// TIA Portal project "2024" (V15.1)

(* hardware
DEVICE "S7300/ET200M station_1"  S7-300 station
   slot 0: "Rail_0"  Rail  6ES7 390-1***0-0AA0
   slot 2: "PLC_1"  CPU 314C-2 PN/DP  6ES7 314-6EH04-0AB0  V3.3
      slot 2: "PROFINET interface_1"  PN-IO
         slot 1: "Port_1"  Port
         slot 2: "Port_2"  Port
      slot 5: "DI 24/DO 16_1"  DI24/DO16
      slot 6: "AI 5/AO 2_1"  AI5/AO2
      slot 7: "Count_1"  Counter
      slot 8: "Positioning_1"  Positioning
   slot 4: "DO 8x24VDC/2A_1"  DO8 x 24VDC / 2A  6ES7 322-1BF01-0AA0
*)

// ===== PLC "PLC_1"  CPU 314C-2 PN/DP =====

VAR_GLOBAL   // PLC tag table "Default tag table"
   "F5" AT %I0.0 : Bool;
   "S3" AT %I0.1 : Bool;
   "S4" AT %I0.2 : Bool;
   "S5" AT %I0.3 : Bool;
   "S6" AT %I0.4 : Bool;
   "S7" AT %I0.5 : Bool;
   "S8" AT %I0.6 : Bool;
   "S9" AT %I0.7 : Bool;
   "S10" AT %I1.0 : Bool;
   "S11" AT %I1.1 : Bool;
   "S12" AT %I1.2 : Bool;
   "BP1" AT %I1.3 : Bool;
   "B1" AT %I1.4 : Bool;
   "B2" AT %I1.5 : Bool;
   "B3" AT %I1.6 : Bool;
   "B11" AT %I1.7 : Bool;
   "B12" AT %I2.0 : Bool;
   "B21" AT %I2.1 : Bool;
   "B22" AT %I2.2 : Bool;
   "B31" AT %I2.3 : Bool;
   "B32" AT %I2.4 : Bool;
   "Reserve1" AT %I2.5 : Bool;
   "Reserve2" AT %I2.6 : Bool;
   "F7" AT %I2.7 : Bool;
   "M11" AT %Q0.0 : Bool;
   "M12" AT %Q0.1 : Bool;
   "M21" AT %Q0.2 : Bool;
   "M22" AT %Q0.3 : Bool;
   "M31" AT %Q0.4 : Bool;
   "M32" AT %Q0.5 : Bool;
   "Reserve3" AT %Q0.6 : Bool;
   "Reserve4" AT %Q0.7 : Bool;
   "P32" AT %Q1.0 : Bool;
   "P33" AT %Q1.1 : Bool;
   "Reserve5" AT %Q1.2 : Bool;
   "P2" AT %Q1.3 : Bool;
   "P3" AT %Q1.4 : Bool;
   "P4" AT %Q1.5 : Bool;
   "P5" AT %Q1.6 : Bool;
   "P6" AT %Q1.7 : Bool;
   "P7" AT %Q2.0 : Bool;
   "P8" AT %Q2.1 : Bool;
   "P10" AT %Q2.2 : Bool;
   "P11" AT %Q2.3 : Bool;
   "P12" AT %Q2.4 : Bool;
   "P13" AT %Q2.5 : Bool;
   "P14" AT %Q2.6 : Bool;
   "P15" AT %Q2.7 : Bool;
END_VAR

DATA_BLOCK "G_Master_DB"   // DB1
{ S7_Optimized_Access := 'FALSE' }
VERSION : 0.1
// stored: InstanceOfName G_Master
"G_Master"
BEGIN
END_DATA_BLOCK

DATA_BLOCK "G_Pulse_DB"   // DB4
{ S7_Optimized_Access := 'FALSE' }
VERSION : 0.1
// stored: InstanceOfName G_Pulse
"G_Pulse"
BEGIN
END_DATA_BLOCK

DATA_BLOCK "G_Manual_DB"   // DB5
{ S7_Optimized_Access := 'FALSE' }
VERSION : 0.1
// stored: InstanceOfName G_Manual
"G_Manual"
BEGIN
END_DATA_BLOCK

DATA_BLOCK "G_Indicator_DB"   // DB6
{ S7_Optimized_Access := 'FALSE' }
VERSION : 0.1
// stored: InstanceOfName G_Indicator
"G_Indicator"
BEGIN
END_DATA_BLOCK

DATA_BLOCK "G_Auto_DB"   // DB13
{ S7_Optimized_Access := 'FALSE' }
VERSION : 0.1
// stored: InstanceOfName G_Auto
"G_Auto"
BEGIN
END_DATA_BLOCK

DATA_BLOCK "G_Output_DB"   // DB14
{ S7_Optimized_Access := 'FALSE' }
VERSION : 0.1
// stored: InstanceOfName G_Output
"G_Output"
BEGIN
END_DATA_BLOCK

FUNCTION_BLOCK "G_Master"   // FB1, FBD
{ S7_Optimized_Access := 'FALSE' }
VERSION : 0.1
   VAR_INPUT
      BP1 : Bool;
      F5 : Bool;
      F7 : Bool;
      S3 : Bool;
      S4 : Bool;
      "G_Auto.X500" : Bool;
      "G_Manual.X300" : Bool;
      Xung : Bool;
   END_VAR
   VAR_OUTPUT
      G_Manual : Bool;
      G_Auto : Bool;
      P3 : Bool;
      P32 : Bool;
   END_VAR
   VAR
      X1 : Bool;
      X2 : Bool;
      X3 : Bool;
      X4 : Bool;
      X5 : Bool;
      MA : Bool;
      MM : Bool;
   END_VAR
BEGIN

REGION Network 1
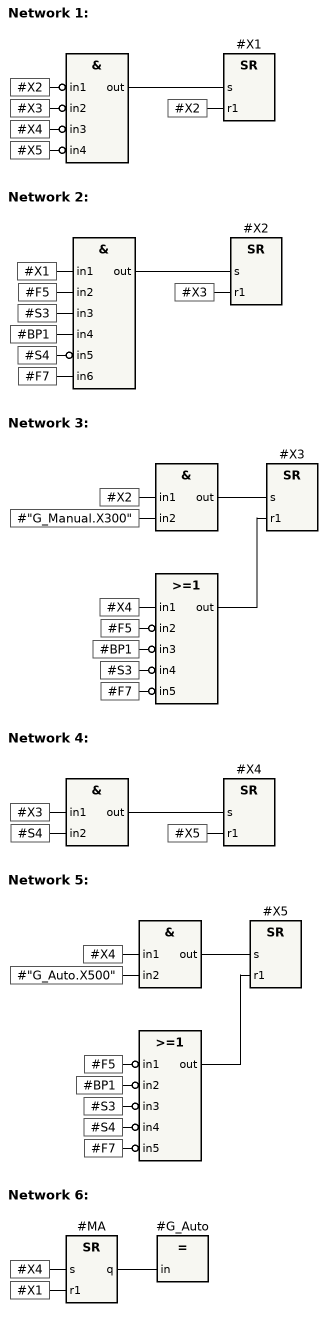
   IF NOT #X2 AND NOT #X3 AND NOT #X4 AND NOT #X5 THEN
       #X1 := TRUE;   // SR flip-flop
   END_IF;
   IF #X2 THEN #X1 := FALSE; END_IF;
END_REGION

REGION Network 2
   IF #X1 AND #F5 AND #S3 AND #BP1 AND NOT #S4 AND #F7 THEN
       #X2 := TRUE;   // SR flip-flop
   END_IF;
   IF #X3 THEN #X2 := FALSE; END_IF;
END_REGION

REGION Network 3
   IF #X2 AND #"G_Manual.X300" THEN
       #X3 := TRUE;   // SR flip-flop
   END_IF;
   IF #X4 OR NOT #F5 OR NOT #BP1 OR NOT #S3 OR NOT #F7 THEN #X3 := FALSE; END_IF;
END_REGION

REGION Network 4
   IF #X3 AND #S4 THEN
       #X4 := TRUE;   // SR flip-flop
   END_IF;
   IF #X5 THEN #X4 := FALSE; END_IF;
END_REGION

REGION Network 5
   IF #X4 AND #"G_Auto.X500" THEN
       #X5 := TRUE;   // SR flip-flop
   END_IF;
   IF NOT #F5 OR NOT #BP1 OR NOT #S3 OR NOT #S4 OR NOT #F7 THEN #X5 := FALSE; END_IF;
END_REGION

REGION Network 6
   IF #X4 THEN
       #MA := TRUE;   // SR flip-flop
   END_IF;
   IF #X1 THEN #MA := FALSE; END_IF;
   #G_Auto := #MA;
END_REGION

REGION Network 7
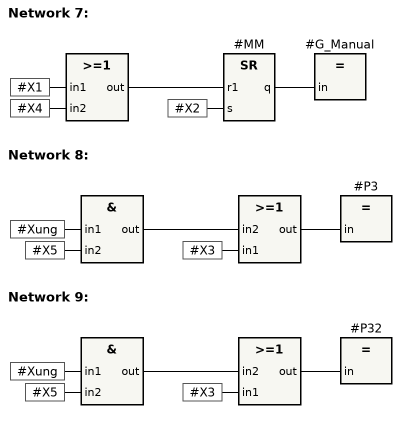
   IF #X2 THEN
       #MM := TRUE;   // SR flip-flop
   END_IF;
   IF #X1 OR #X4 THEN #MM := FALSE; END_IF;
   #G_Manual := #MM;
END_REGION

REGION Network 8
   #P3 := (#Xung AND #X5) OR #X3;
END_REGION

REGION Network 9
   #P32 := (#Xung AND #X5) OR #X3;
END_REGION
END_FUNCTION_BLOCK

FUNCTION_BLOCK "G_Pulse"   // FB2, FBD
{ S7_Optimized_Access := 'FALSE' }
VERSION : 0.1
   VAR_OUTPUT
      Pulse : Bool;
   END_VAR
   VAR
      X100 : Bool;
      X101 : Bool;
   END_VAR
BEGIN

REGION Network 1
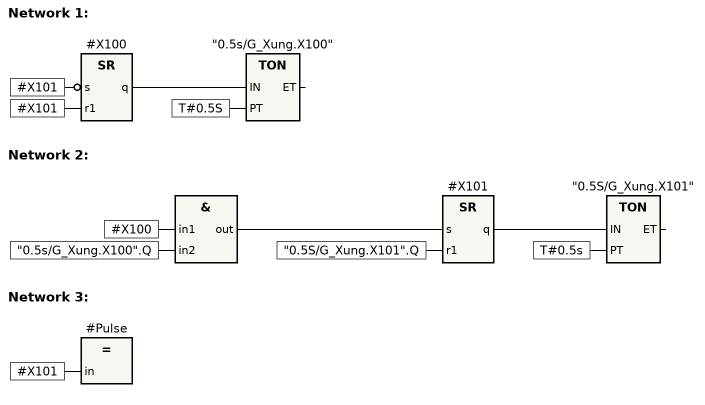
   IF NOT #X101 THEN
       #X100 := TRUE;   // SR flip-flop
   END_IF;
   IF #X101 THEN #X100 := FALSE; END_IF;
   "0.5s/G_Xung.X100".TON(IN := #X100, PT := T#0.5S);
END_REGION

REGION Network 2
   IF #X100 AND "0.5s/G_Xung.X100".Q THEN
       #X101 := TRUE;   // SR flip-flop
   END_IF;
   IF "0.5S/G_Xung.X101".Q THEN #X101 := FALSE; END_IF;
   "0.5S/G_Xung.X101".TON(IN := #X101, PT := T#0.5s);
END_REGION

REGION Network 3
   #Pulse := #X101;
END_REGION
END_FUNCTION_BLOCK

FUNCTION_BLOCK "G_Manual"   // FB3, FBD
{ S7_Optimized_Access := 'FALSE' }
VERSION : 0.1
   VAR_INPUT
      G_Manual : Bool;
      S4 : Bool;
      S6 : Bool;
      S7 : Bool;
      S8 : Bool;
      S9 : Bool;
      S10 : Bool;
      S11 : Bool;
   END_VAR
   VAR_OUTPUT
      M11 : Bool;
      M12 : Bool;
      M21 : Bool;
      M22 : Bool;
      M31 : Bool;
      M32 : Bool;
   END_VAR
   VAR
      X300 : Bool;
      X301 : Bool;
   END_VAR
BEGIN

REGION Network 1
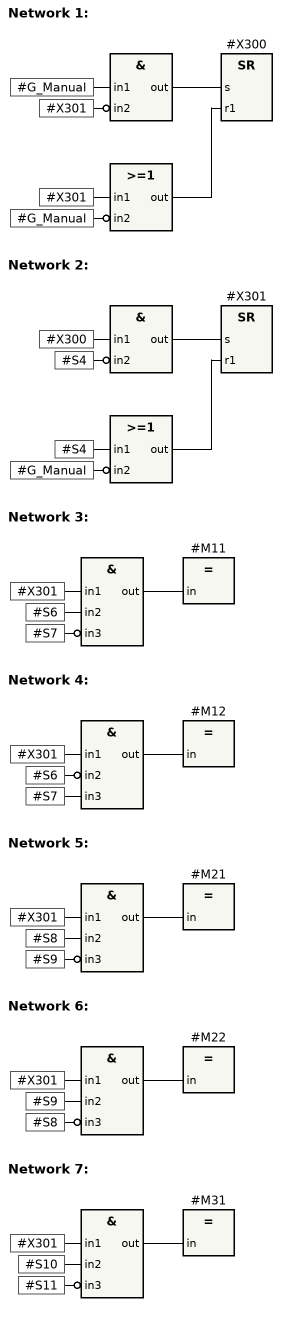
   IF #G_Manual AND NOT #X301 THEN
       #X300 := TRUE;   // SR flip-flop
   END_IF;
   IF #X301 OR NOT #G_Manual THEN #X300 := FALSE; END_IF;
END_REGION

REGION Network 2
   IF #X300 AND NOT #S4 THEN
       #X301 := TRUE;   // SR flip-flop
   END_IF;
   IF #S4 OR NOT #G_Manual THEN #X301 := FALSE; END_IF;
END_REGION

REGION Network 3
   #M11 := #X301 AND #S6 AND NOT #S7;
END_REGION

REGION Network 4
   #M12 := #X301 AND NOT #S6 AND #S7;
END_REGION

REGION Network 5
   #M21 := #X301 AND #S8 AND NOT #S9;
END_REGION

REGION Network 6
   #M22 := #X301 AND #S9 AND NOT #S8;
END_REGION

REGION Network 7
   #M31 := #X301 AND #S10 AND NOT #S11;
END_REGION

REGION Network 8
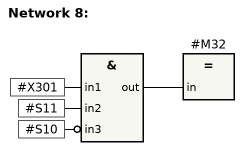
   #M32 := #X301 AND #S11 AND NOT #S10;
END_REGION
END_FUNCTION_BLOCK

FUNCTION_BLOCK "G_Indicator"   // FB4, FBD
{ S7_Optimized_Access := 'FALSE' }
VERSION : 0.1
   VAR_INPUT
      S3 : Bool;
      S12 : Bool;
      F7 : Bool;
      BP1 : Bool;
      B1 : Bool;
      B2 : Bool;
      B3 : Bool;
      B11 : Bool;
      B12 : Bool;
      B21 : Bool;
      B22 : Bool;
      B31 : Bool;
      B32 : Bool;
   END_VAR
   VAR_OUTPUT
      P2 : Bool;
      P3 : Bool;
      P4 : Bool;
      P5 : Bool;
      P6 : Bool;
      P7 : Bool;
      P8 : Bool;
      P10 : Bool;
      P11 : Bool;
      P12 : Bool;
      P13 : Bool;
      P14 : Bool;
      P15 : Bool;
      P32 : Bool;
      P33 : Bool;
   END_VAR
   VAR
      X200 : Bool;
      X201 : Bool;
   END_VAR
BEGIN

REGION Network 1
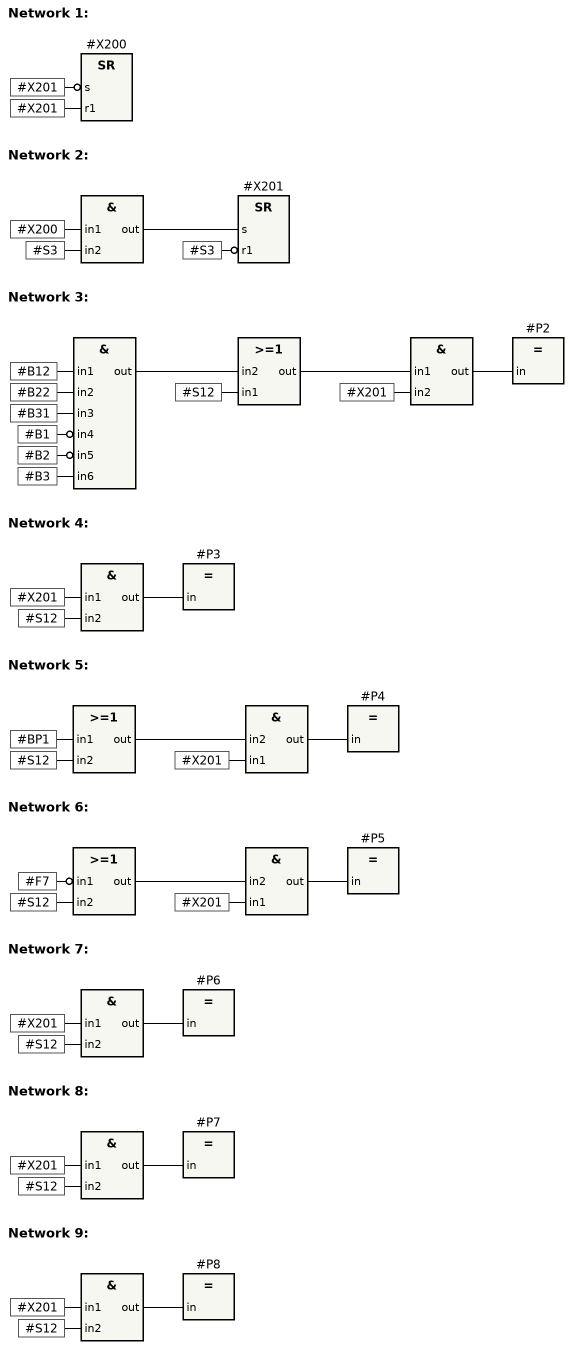
   IF NOT #X201 THEN
       #X200 := TRUE;   // SR flip-flop
   END_IF;
   IF #X201 THEN #X200 := FALSE; END_IF;
END_REGION

REGION Network 2
   IF #X200 AND #S3 THEN
       #X201 := TRUE;   // SR flip-flop
   END_IF;
   IF NOT #S3 THEN #X201 := FALSE; END_IF;
END_REGION

REGION Network 3
   #P2 := ((#B12 AND #B22 AND #B31 AND NOT #B1 AND NOT #B2 AND #B3) OR #S12) AND #X201;
END_REGION

REGION Network 4
   #P3 := #X201 AND #S12;
END_REGION

REGION Network 5
   #P4 := (#BP1 OR #S12) AND #X201;
END_REGION

REGION Network 6
   #P5 := (NOT #F7 OR #S12) AND #X201;
END_REGION

REGION Network 7
   #P6 := #X201 AND #S12;
END_REGION

REGION Network 8
   #P7 := #X201 AND #S12;
END_REGION

REGION Network 9
   #P8 := #X201 AND #S12;
END_REGION

REGION Network 10
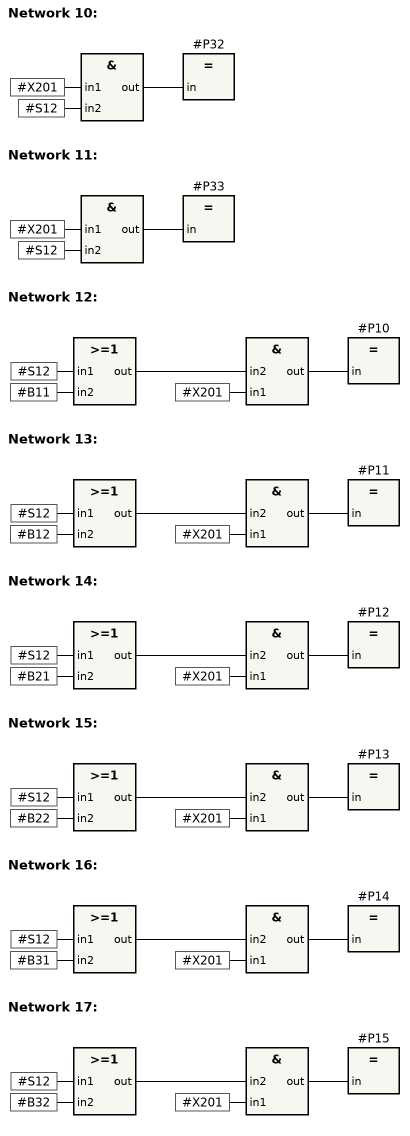
   #P32 := #X201 AND #S12;
END_REGION

REGION Network 11
   #P33 := #X201 AND #S12;
END_REGION

REGION Network 12
   #P10 := (#S12 OR #B11) AND #X201;
END_REGION

REGION Network 13
   #P11 := (#S12 OR #B12) AND #X201;
END_REGION

REGION Network 14
   #P12 := (#S12 OR #B21) AND #X201;
END_REGION

REGION Network 15
   #P13 := (#S12 OR #B22) AND #X201;
END_REGION

REGION Network 16
   #P14 := (#S12 OR #B31) AND #X201;
END_REGION

REGION Network 17
   #P15 := (#S12 OR #B32) AND #X201;
END_REGION
END_FUNCTION_BLOCK

FUNCTION_BLOCK "G_Auto"   // FB5, FBD
{ S7_Optimized_Access := 'FALSE' }
VERSION : 0.1
   VAR_INPUT
      "G_Master.X1" : Bool;
      G_Auto : Bool;
      S5 : Bool;
      B1 : Bool;
      B2 : Bool;
      B3 : Bool;
      B11 : Bool;
      B12 : Bool;
      B21 : Bool;
      B22 : Bool;
      B31 : Bool;
      B32 : Bool;
   END_VAR
   VAR_OUTPUT
      P6 : Bool;
      P7 : Bool;
      P8 : Bool;
      P33 : Bool;
      M11 : Bool;
      M12 : Bool;
      M21 : Bool;
      M22 : Bool;
      M31 : Bool;
      M32 : Bool;
   END_VAR
   VAR
      X500 : Bool;
      X501 : Bool;
      X502 : Bool;
      X503 : Bool;
      X503a : Bool;
      X504 : Bool;
      X504a : Bool;
      X505 : Bool;
      X506 : Bool;
      X507 : Bool;
      X508 : Bool;
      M6 : Bool;
      M7 : Bool;
   END_VAR
BEGIN

REGION Network 1
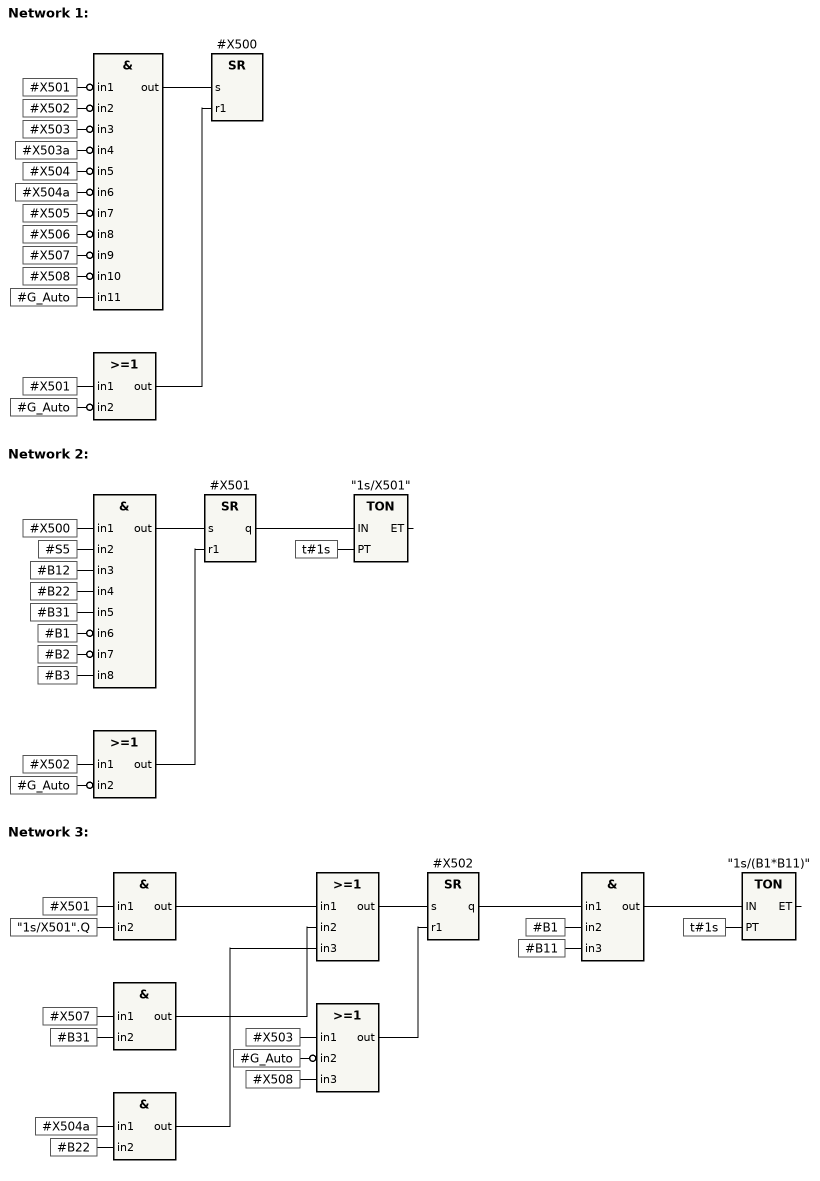
   IF NOT #X501 AND NOT #X502 AND NOT #X503 AND NOT #X503a AND NOT #X504 AND NOT #X504a AND NOT #X505 AND NOT #X506 AND NOT #X507 AND NOT #X508 AND #G_Auto THEN
       #X500 := TRUE;   // SR flip-flop
   END_IF;
   IF #X501 OR NOT #G_Auto THEN #X500 := FALSE; END_IF;
END_REGION

REGION Network 2
   IF #X500 AND #S5 AND #B12 AND #B22 AND #B31 AND NOT #B1 AND NOT #B2 AND #B3 THEN
       #X501 := TRUE;   // SR flip-flop
   END_IF;
   IF #X502 OR NOT #G_Auto THEN #X501 := FALSE; END_IF;
   "1s/X501".TON(IN := #X501, PT := t#1s);
END_REGION

REGION Network 3
   IF (#X501 AND "1s/X501".Q) OR (#X507 AND #B31) OR (#X504a AND #B22) THEN
       #X502 := TRUE;   // SR flip-flop
   END_IF;
   IF #X503 OR NOT #G_Auto OR #X508 THEN #X502 := FALSE; END_IF;
   "1s/(B1*B11)".TON(IN := #X502 AND #B1 AND #B11, PT := t#1s);
END_REGION

REGION Network 4
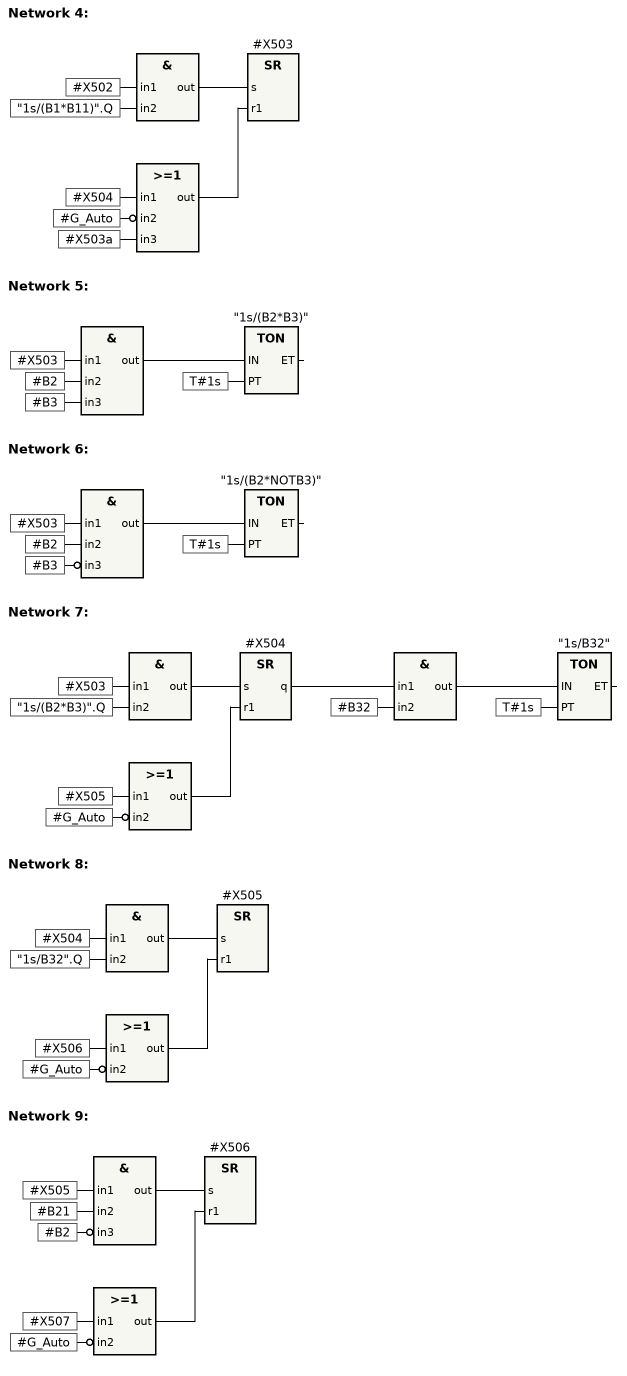
   IF #X502 AND "1s/(B1*B11)".Q THEN
       #X503 := TRUE;   // SR flip-flop
   END_IF;
   IF #X504 OR NOT #G_Auto OR #X503a THEN #X503 := FALSE; END_IF;
END_REGION

REGION Network 5
   "1s/(B2*B3)".TON(IN := #X503 AND #B2 AND #B3, PT := T#1s);
END_REGION

REGION Network 6
   "1s/(B2*NOTB3)".TON(IN := #X503 AND #B2 AND NOT #B3, PT := T#1s);
END_REGION

REGION Network 7
   IF #X503 AND "1s/(B2*B3)".Q THEN
       #X504 := TRUE;   // SR flip-flop
   END_IF;
   IF #X505 OR NOT #G_Auto THEN #X504 := FALSE; END_IF;
   "1s/B32".TON(IN := #X504 AND #B32, PT := T#1s);
END_REGION

REGION Network 8
   IF #X504 AND "1s/B32".Q THEN
       #X505 := TRUE;   // SR flip-flop
   END_IF;
   IF #X506 OR NOT #G_Auto THEN #X505 := FALSE; END_IF;
END_REGION

REGION Network 9
   IF #X505 AND #B21 AND NOT #B2 THEN
       #X506 := TRUE;   // SR flip-flop
   END_IF;
   IF #X507 OR NOT #G_Auto THEN #X506 := FALSE; END_IF;
END_REGION

REGION Network 10
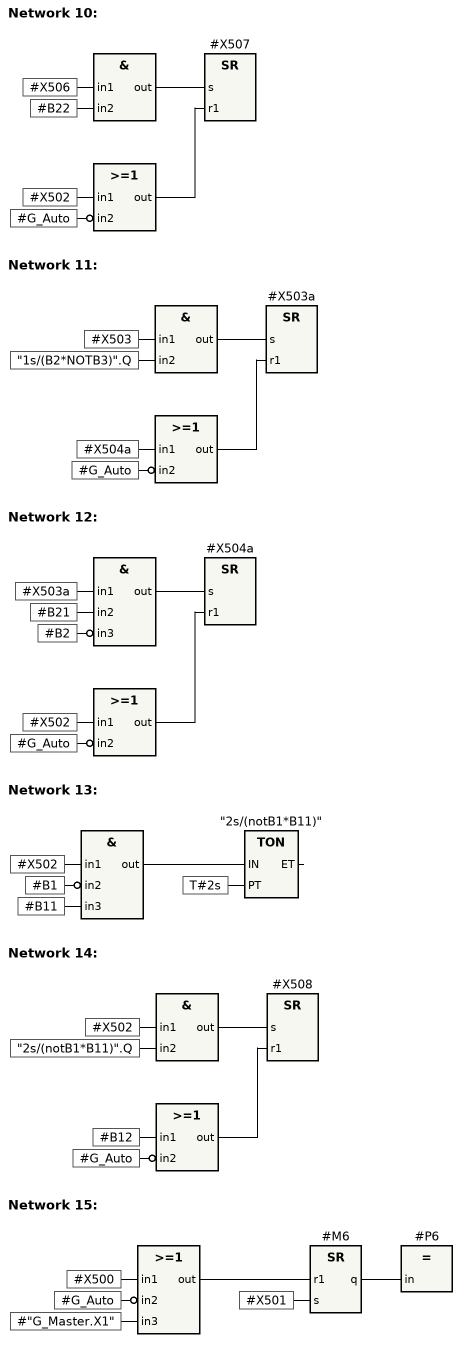
   IF #X506 AND #B22 THEN
       #X507 := TRUE;   // SR flip-flop
   END_IF;
   IF #X502 OR NOT #G_Auto THEN #X507 := FALSE; END_IF;
END_REGION

REGION Network 11
   IF #X503 AND "1s/(B2*NOTB3)".Q THEN
       #X503a := TRUE;   // SR flip-flop
   END_IF;
   IF #X504a OR NOT #G_Auto THEN #X503a := FALSE; END_IF;
END_REGION

REGION Network 12
   IF #X503a AND #B21 AND NOT #B2 THEN
       #X504a := TRUE;   // SR flip-flop
   END_IF;
   IF #X502 OR NOT #G_Auto THEN #X504a := FALSE; END_IF;
END_REGION

REGION Network 13
   "2s/(notB1*B11)".TON(IN := #X502 AND NOT #B1 AND #B11, PT := T#2s);
END_REGION

REGION Network 14
   IF #X502 AND "2s/(notB1*B11)".Q THEN
       #X508 := TRUE;   // SR flip-flop
   END_IF;
   IF #B12 OR NOT #G_Auto THEN #X508 := FALSE; END_IF;
END_REGION

REGION Network 15
   IF #X501 THEN
       #M6 := TRUE;   // SR flip-flop
   END_IF;
   IF #X500 OR NOT #G_Auto OR #"G_Master.X1" THEN #M6 := FALSE; END_IF;
   #P6 := #M6;
END_REGION

REGION Network 16
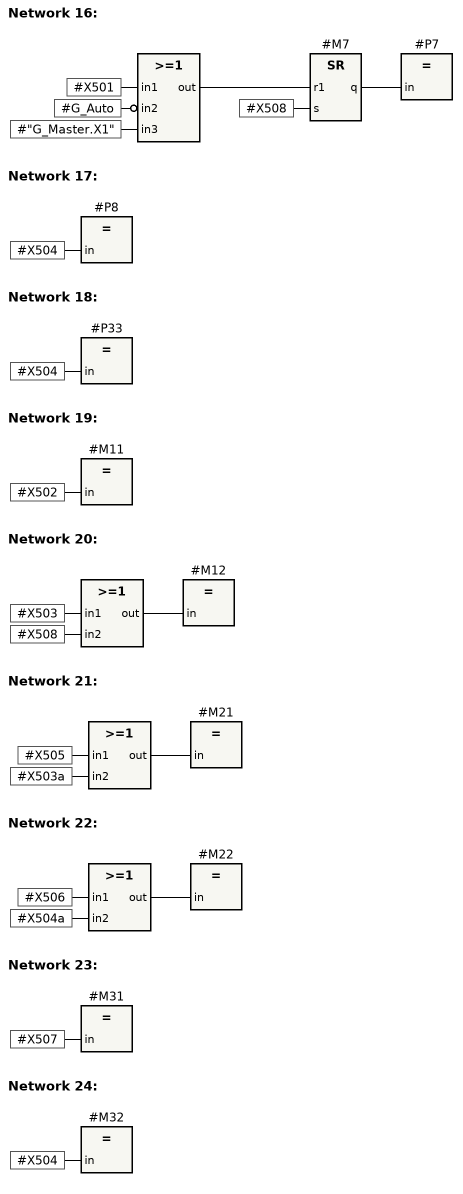
   IF #X508 THEN
       #M7 := TRUE;   // SR flip-flop
   END_IF;
   IF #X501 OR NOT #G_Auto OR #"G_Master.X1" THEN #M7 := FALSE; END_IF;
   #P7 := #M7;
END_REGION

REGION Network 17
   #P8 := #X504;
END_REGION

REGION Network 18
   #P33 := #X504;
END_REGION

REGION Network 19
   #M11 := #X502;
END_REGION

REGION Network 20
   #M12 := #X503 OR #X508;
END_REGION

REGION Network 21
   #M21 := #X505 OR #X503a;
END_REGION

REGION Network 22
   #M22 := #X506 OR #X504a;
END_REGION

REGION Network 23
   #M31 := #X507;
END_REGION

REGION Network 24
   #M32 := #X504;
END_REGION
END_FUNCTION_BLOCK

FUNCTION_BLOCK "G_Output"   // FB6, FBD
{ S7_Optimized_Access := 'FALSE' }
VERSION : 0.1
   VAR_INPUT
      M11_M : Bool;
      M12_M : Bool;
      M21_M : Bool;
      M22_M : Bool;
      M31_M : Bool;
      M32_M : Bool;
      M11_A : Bool;
      M12_A : Bool;
      M21_A : Bool;
      M22_A : Bool;
      M31_A : Bool;
      M32_A : Bool;
      P3_M : Bool;
      P32_M : Bool;
      P6_A : Bool;
      P7_A : Bool;
      P8_A : Bool;
      P33_A : Bool;
      P3_I : Bool;
      P6_I : Bool;
      P7_I : Bool;
      P8_I : Bool;
      P33_I : Bool;
      P32_I : Bool;
   END_VAR
   VAR_OUTPUT
      M11 : Bool;
      M12 : Bool;
      M21 : Bool;
      M22 : Bool;
      M31 : Bool;
      M32 : Bool;
      P3 : Bool;
      P6 : Bool;
      P7 : Bool;
      P8 : Bool;
      P33 : Bool;
      P32 : Bool;
   END_VAR
BEGIN

REGION Network 1
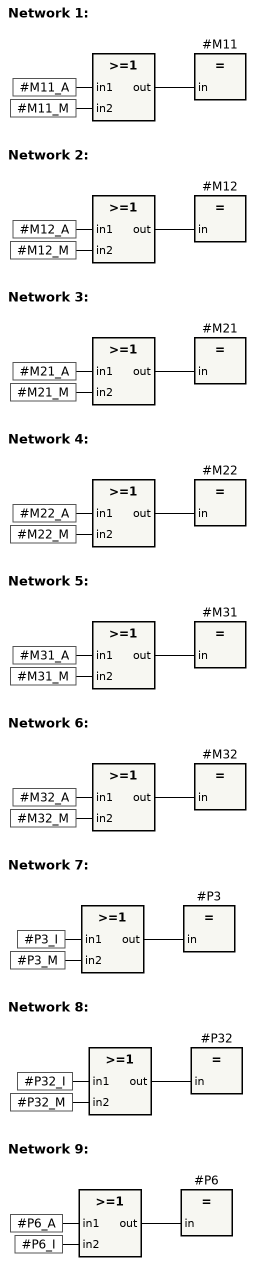
   #M11 := #M11_A OR #M11_M;
END_REGION

REGION Network 2
   #M12 := #M12_A OR #M12_M;
END_REGION

REGION Network 3
   #M21 := #M21_A OR #M21_M;
END_REGION

REGION Network 4
   #M22 := #M22_A OR #M22_M;
END_REGION

REGION Network 5
   #M31 := #M31_A OR #M31_M;
END_REGION

REGION Network 6
   #M32 := #M32_A OR #M32_M;
END_REGION

REGION Network 7
   #P3 := #P3_I OR #P3_M;
END_REGION

REGION Network 8
   #P32 := #P32_I OR #P32_M;
END_REGION

REGION Network 9
   #P6 := #P6_A OR #P6_I;
END_REGION

REGION Network 10
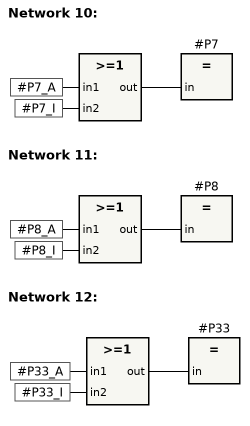
   #P7 := #P7_A OR #P7_I;
END_REGION

REGION Network 11
   #P8 := #P8_A OR #P8_I;
END_REGION

REGION Network 12
   #P33 := #P33_A OR #P33_I;
END_REGION
END_FUNCTION_BLOCK

ORGANIZATION_BLOCK "Main"   // OB1, FBD
TITLE = "Main Program Sweep (Cycle)"
{ S7_Optimized_Access := 'FALSE' }
VERSION : 0.1
   VAR_TEMP
      OB1_EV_CLASS : Byte;   // Bits 0-3 = 1 (Coming event), Bits 4-7 = 1 (Event class 1)
      OB1_SCAN_1 : Byte;   // 1 (Cold restart scan 1 of OB 1), 3 (Scan 2-n of OB 1)
      OB1_PRIORITY : Byte;   // Priority of OB Execution
      OB1_OB_NUMBR : Byte;   // 1 (Organization block 1, OB1)
      OB1_RESERVED_1 : Byte;   // Reserved for system
      OB1_RESERVED_2 : Byte;   // Reserved for system
      OB1_PREV_CYCLE : Int;   // Cycle time of previous OB1 scan (milliseconds)
      OB1_MIN_CYCLE : Int;   // Minimum cycle time of OB1 (milliseconds)
      OB1_MAX_CYCLE : Int;   // Maximum cycle time of OB1 (milliseconds)
      OB1_DATE_TIME : Date_And_Time;   // Date and time OB1 started
   END_VAR
BEGIN

REGION Network 1
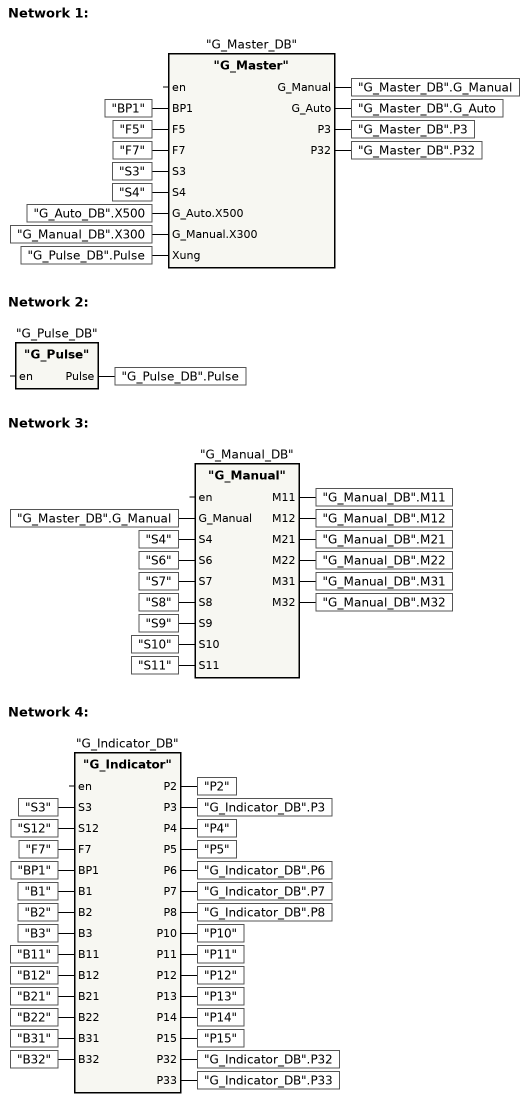
   "G_Master_DB"(BP1 := "BP1",   // "G_Master"
                 F5 := "F5",
                 F7 := "F7",
                 S3 := "S3",
                 S4 := "S4",
                 "G_Auto.X500" := "G_Auto_DB".X500,
                 "G_Manual.X300" := "G_Manual_DB".X300,
                 Xung := "G_Pulse_DB".Pulse,
                 G_Manual => "G_Master_DB".G_Manual,
                 G_Auto => "G_Master_DB".G_Auto,
                 P3 => "G_Master_DB".P3,
                 P32 => "G_Master_DB".P32);
END_REGION

REGION Network 2
   "G_Pulse_DB"(Pulse => "G_Pulse_DB".Pulse);   // "G_Pulse"
END_REGION

REGION Network 3
   "G_Manual_DB"(G_Manual := "G_Master_DB".G_Manual,   // "G_Manual"
                 S4 := "S4",
                 S6 := "S6",
                 S7 := "S7",
                 S8 := "S8",
                 S9 := "S9",
                 S10 := "S10",
                 S11 := "S11",
                 M11 => "G_Manual_DB".M11,
                 M12 => "G_Manual_DB".M12,
                 M21 => "G_Manual_DB".M21,
                 M22 => "G_Manual_DB".M22,
                 M31 => "G_Manual_DB".M31,
                 M32 => "G_Manual_DB".M32);
END_REGION

REGION Network 4
   "G_Indicator_DB"(S3 := "S3",   // "G_Indicator"
                    S12 := "S12",
                    F7 := "F7",
                    BP1 := "BP1",
                    B1 := "B1",
                    B2 := "B2",
                    B3 := "B3",
                    B11 := "B11",
                    B12 := "B12",
                    B21 := "B21",
                    B22 := "B22",
                    B31 := "B31",
                    B32 := "B32",
                    P2 => "P2",
                    P3 => "G_Indicator_DB".P3,
                    P4 => "P4",
                    P5 => "P5",
                    P6 => "G_Indicator_DB".P6,
                    P7 => "G_Indicator_DB".P7,
                    P8 => "G_Indicator_DB".P8,
                    P10 => "P10",
                    P11 => "P11",
                    P12 => "P12",
                    P13 => "P13",
                    P14 => "P14",
                    P15 => "P15",
                    P32 => "G_Indicator_DB".P32,
                    P33 => "G_Indicator_DB".P33);
END_REGION

REGION Network 5
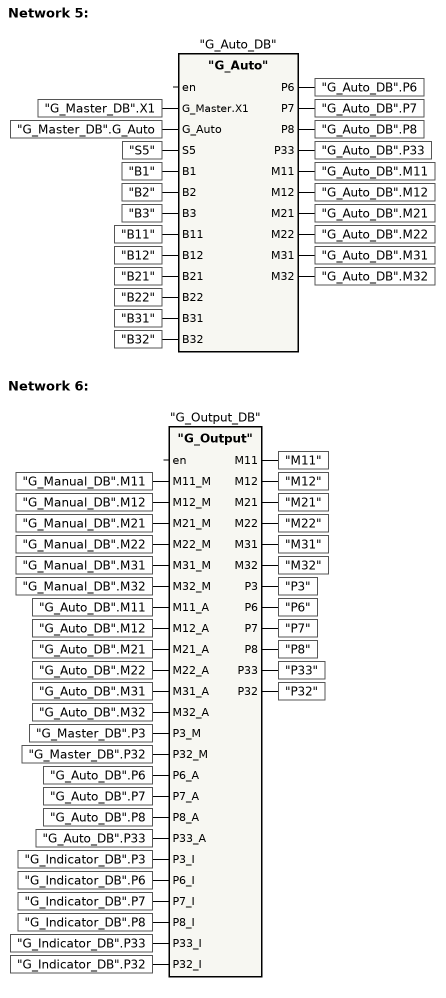
   "G_Auto_DB"("G_Master.X1" := "G_Master_DB".X1,   // "G_Auto"
               G_Auto := "G_Master_DB".G_Auto,
               S5 := "S5",
               B1 := "B1",
               B2 := "B2",
               B3 := "B3",
               B11 := "B11",
               B12 := "B12",
               B21 := "B21",
               B22 := "B22",
               B31 := "B31",
               B32 := "B32",
               P6 => "G_Auto_DB".P6,
               P7 => "G_Auto_DB".P7,
               P8 => "G_Auto_DB".P8,
               P33 => "G_Auto_DB".P33,
               M11 => "G_Auto_DB".M11,
               M12 => "G_Auto_DB".M12,
               M21 => "G_Auto_DB".M21,
               M22 => "G_Auto_DB".M22,
               M31 => "G_Auto_DB".M31,
               M32 => "G_Auto_DB".M32);
END_REGION

REGION Network 6
   "G_Output_DB"(M11_M := "G_Manual_DB".M11,   // "G_Output"
                 M12_M := "G_Manual_DB".M12,
                 M21_M := "G_Manual_DB".M21,
                 M22_M := "G_Manual_DB".M22,
                 M31_M := "G_Manual_DB".M31,
                 M32_M := "G_Manual_DB".M32,
                 M11_A := "G_Auto_DB".M11,
                 M12_A := "G_Auto_DB".M12,
                 M21_A := "G_Auto_DB".M21,
                 M22_A := "G_Auto_DB".M22,
                 M31_A := "G_Auto_DB".M31,
                 M32_A := "G_Auto_DB".M32,
                 P3_M := "G_Master_DB".P3,
                 P32_M := "G_Master_DB".P32,
                 P6_A := "G_Auto_DB".P6,
                 P7_A := "G_Auto_DB".P7,
                 P8_A := "G_Auto_DB".P8,
                 P33_A := "G_Auto_DB".P33,
                 P3_I := "G_Indicator_DB".P3,
                 P6_I := "G_Indicator_DB".P6,
                 P7_I := "G_Indicator_DB".P7,
                 P8_I := "G_Indicator_DB".P8,
                 P33_I := "G_Indicator_DB".P33,
                 P32_I := "G_Indicator_DB".P32,
                 M11 => "M11",
                 M12 => "M12",
                 M21 => "M21",
                 M22 => "M22",
                 M31 => "M31",
                 M32 => "M32",
                 P3 => "P3",
                 P6 => "P6",
                 P7 => "P7",
                 P8 => "P8",
                 P33 => "P33",
                 P32 => "P32");
END_REGION
END_ORGANIZATION_BLOCK